# B&R Automation Studio project PO3
Automation Studio 4.5.2.102

## Configuration Real

### Hardware
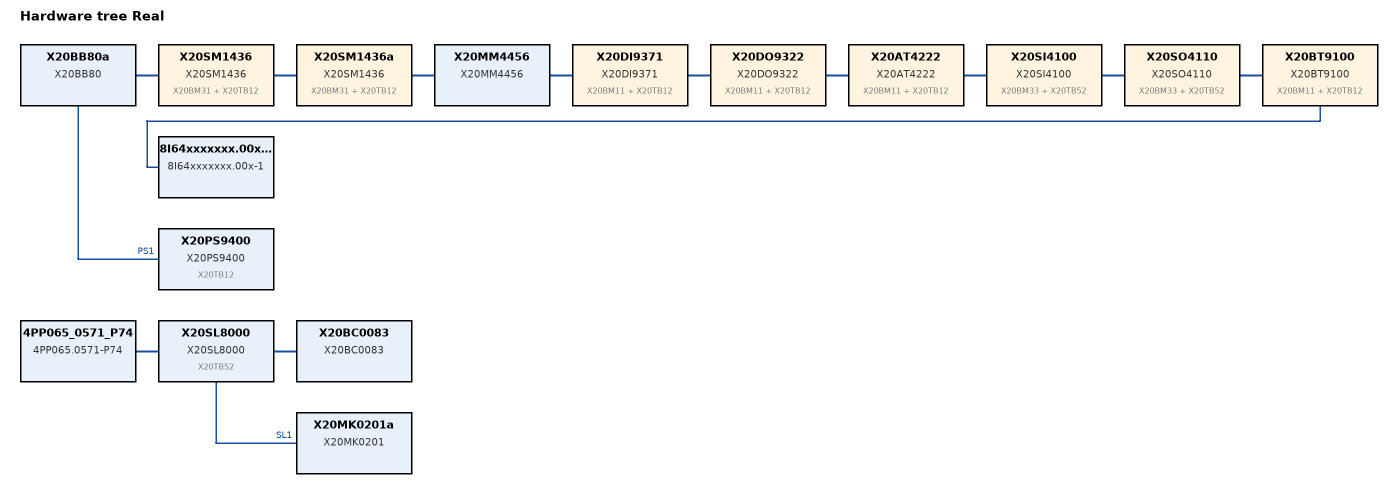
```
4PP065_0571_P74 : 4PP065.0571-P74 v1.1.2.0
  Connector IF4:
    EplInterfaceRedundant = 0
    EplEthInterfaceRedundant = 0
  Connector IF5:
    ActivateDevice = 1
    Mode = Manual
    InternetAddress = 10.0.1.10
    SubnetMask = 255.255.255.0
  ConfigurationID = LabBR
  TimerDeviceType = EPLX2X
  TimerDevice = 4PP065_0571_P74.IF4
  TaskClassIdleTime = 2000
  Cyclic1Duration = 2000
  Cyclic1Tolerance = 0
  Cyclic1Output = 1
  Cyclic3Tolerance = 0
  VcObjectName = Visu
8I64xxxxxxx.00x-1 : 8I64xxxxxxx.00x-1 v1.3.9.1  [X2X1 -> X20BT9100.X2X1 [Cable Type=X2XCable, Length=10, Version=1.0.0.2]]
  BothEndSwitchesAreNormallyOpen_r1 = on
  QuickStopIsNormallyOpen_r1 = on
X20AT4222 : X20AT4222 v1.2.3.0  [SS1 -> X20TB12f.SS; SL -> X20BM11c.SL1]
X20BB80a : X20BB80 v1.0.2.0
X20BC0083 : X20BC0083 v2.7.0.0  [PLK1 -> X20SL8000.PLK2 (NodeNumber=2) [Cable Type=PowerlinkCable, Length=10, Version=1.0.0.2]; SL -> X20BB80a.SL1]
X20BM11a : X20BM11 v1.0.0.1  [X2X1 -> X20MM4456.X2X2]
X20BM11b : X20BM11 v1.0.0.1  [X2X1 -> X20BM11a.X2X2]
X20BM11c : X20BM11 v1.0.0.1  [X2X1 -> X20BM11b.X2X2]
X20BM11d : X20BM11 v1.0.0.1  [X2X1 -> X20BM33b.X2X2]
X20BM31a : X20BM31 v1.0.0.1  [X2X1 -> X20BB80a.IF1]
X20BM31b : X20BM31 v1.0.0.1  [X2X1 -> X20BM31a.X2X2]
X20BM33a : X20BM33 v1.0.0.4  [X2X1 -> X20BM11c.X2X2]
X20BM33b : X20BM33 v1.0.0.4  [X2X1 -> X20BM33a.X2X2]
X20BT9100 : X20BT9100 v1.0.3.0  [SS1 -> X20TB12g.SS; SL -> X20BM11d.SL1]
X20DI9371 : X20DI9371 v1.0.2.0  [SS1 -> X20TB12d.SS; SL -> X20BM11a.SL1]
X20DO9322 : X20DO9322 v1.0.3.0  [SS1 -> X20TB12e.SS; SL -> X20BM11b.SL1]
X20MK0201a : X20MK0201 v1.0.0.0  [SL -> X20SL8000.SL1]
X20MM4456 : X20MM4456 v1.1.5.0  [X2X1 -> X20BM31b.X2X2]
X20PS9400 : X20PS9400 v1.0.2.4  [SS1 -> X20TB12b.SS; PS -> X20BB80a.PS1]
X20SI4100 : X20SI4100 v1.10.1.1  [SS1 -> X20TB52b.SS; SL -> X20BM33a.SL1]
X20SL8000 : X20SL8000 v1.6.5.1  [PLK1 -> 4PP065_0571_P74.IF4 (NodeNumber=1) [Cable Type=PowerlinkCable, Length=10, Version=1.0.0.2]; PLK2 -> X20BC0083.PLK1 (NodeNumber=1) [Cable Type=PowerlinkCable, Length=10, Version=1.0.0.2]; SS1 -> X20TB52a.SS]
  SafeProject = SafeLOGIC-1
X20SM1436 : X20SM1436 v1.4.2.1  [SS1 -> X20TB12a.SS; SL -> X20BM31a.SL1]
X20SM1436a : X20SM1436 v1.4.2.1  [SS1 -> X20TB12c.SS; SL -> X20BM31b.SL1]
X20SO4110 : X20SO4110 v1.10.1.1  [SS1 -> X20TB52c.SS; SL -> X20BM33b.SL1]
  SafeLogicID = 2
  SafeModuleID = 3
X20TB12a : X20TB12 v1.0.0.0
X20TB12b : X20TB12 v1.0.0.0
X20TB12c : X20TB12 v1.0.0.0
X20TB12d : X20TB12 v1.0.0.0
X20TB12e : X20TB12 v1.0.0.0
X20TB12f : X20TB12 v1.0.0.0
X20TB12g : X20TB12 v1.0.0.0
X20TB52a : X20TB52 v1.0.0.1
X20TB52b : X20TB52 v1.0.0.1
X20TB52c : X20TB52 v1.0.0.1
```

### IoMap.iom - 4PP065_0571_P74/IoMap.iom
```iecst
VAR_CONFIG
	Cyclic#1.gAxis03_DrvIf.iLifeCnt AT %IB."8I64xxxxxxx.00x-1".SDC_LifeCnt;
	Cyclic#1.gAxis03_DrvIf.iDrvOK AT %IX."8I64xxxxxxx.00x-1".ETAD_Input_Bool_02;
	Cyclic#1.gAxis03_DrvIf.oSetTime AT %QW."8I64xxxxxxx.00x-1".SDC_SetTime;
	Cyclic#1.gAxis03_DrvIf.oSetPos AT %QW."8I64xxxxxxx.00x-1".LFRD_Output;
	Cyclic#1.gAxis03_DiDoIf.iLifeCntDriveReady AT %IB."8I64xxxxxxx.00x-1".SDC_LifeCnt;
	Cyclic#1.gAxis03_DiDoIf.iLifeCntDriveEnable AT %IB."8I64xxxxxxx.00x-1".SDC_LifeCnt;
	Cyclic#1.gAxis03_DiDoIf.oDriveEnable AT %QX."8I64xxxxxxx.00x-1".CMDD_Output_Bool_00;
	Cyclic#1.gAxis03_ModuleOk AT %QX."8I64xxxxxxx.00x-1".CMDD_Output_Bool_01;
	Cyclic#1.gAxis03_ModuleOk AT %QX."8I64xxxxxxx.00x-1".CMDD_Output_Bool_02;
	Cyclic#1.gAxis03_ModuleOk AT %IX."8I64xxxxxxx.00x-1".ModuleOk;
	Cyclic#1.gAxis03_DiDoIf.oDriveEnable AT %QX."8I64xxxxxxx.00x-1".CMDD_Output_Bool_03;
	Cyclic#1.gAxis03_DiDoIf.iDriveReady AT %IX."8I64xxxxxxx.00x-1".ETAD_Input_Bool_02;
	::SDCAxisCtr:pwm_period AT %QW."X20MM4456".PeriodDurationPWM;
	::SDCAxisCtr:coil_pwm_value AT %QW."X20MM4456".PulseWidthCurrentPWM04;
	::SDCAxisCtr:axis_X.pwm_value AT %QW."X20MM4456".PulseWidthCurrentPWM01;
	::SDCAxisCtr:axis_X.reset_error AT %QX."X20MM4456".ClearError01;
	::SDCAxisCtr:axis_X.reset_counter AT %QX."X20MM4456".ResetCounter01;
	::SDCAxisCtr:axis_X.counter AT %IW."X20MM4456".Counter01;
	::SDCAxisCtr:coil_powered AT %IX."X20DI9371".DigitalInput01;
	::SDCAxisCtr:axis_X.endswitch_a_reached AT %IX."X20MM4456".StatusInput03;
	::SDCAxisCtr:axis_X.endswitch_b_reached AT %IX."X20MM4456".StatusInput04;
	::SDCAxisCtr:posEnable.enable AT %IX."X20DI9371".DigitalInput02; (*Insert your comment here...*)
	::SDCAxisCtr:posEnableRight.enable AT %IX."X20DI9371".DigitalInput03; (*Insert your comment here...*)
END_VAR
```

## Logical view

### Program Logical/Libraries/Library

#### FB_Axis.c
```c
#include <bur/plctypes.h>
#ifdef __cplusplus
	extern "C"
	{
#endif
	#include "Library.h"
#ifdef __cplusplus
	};
#endif
/* TODO: Add your comment here */
void FB_Axis(struct FB_Axis* inst)
{
	if (inst->endswitch_a_reached == 1 )
	{
		inst->dir = 1;
	}
	if (inst->endswitch_b_reached == 1 )
	{
		inst->dir = 0;
	}

	if(inst->dir == 1)
	{
		//inst->reset_counter = 0;
		inst->u = -inst->u;
		inst->pwm_value = (inst->u/24.0) * 32767;
	}
	if(inst->dir == 0)
	{
		//inst->reset_counter = 0;
		inst->pwm_value = (inst->u/24.0) * 32767;
	}
	if (inst->i == 1000)
	{
		inst->speed = (inst->counter - inst->last_counter)/2;
		inst->last_counter = inst->counter;
		inst->i = 0;
	}
	inst->spid = inst->speed;
	inst->i++;
}
```

### Program Logical/SDCAxisCtrl_X

#### Variables.var
```iecst
VAR
	min_task : INT := 7000;
	desired_speed : INT := 0;
	axis_X : FB_Axis;
	coil_powered : BOOL := FALSE;
	coil_pwm_value : {REDUND_UNREPLICABLE} INT := 200;
	fb_controller : FB_Controller;
	pwm_period : {REDUND_UNREPLICABLE} UINT := 200;
	Already_Homed : BOOL := FALSE;
	k : INT := 0;
	reset : BOOL := FALSE;
	posEnable : Pos := (0);
	posEnableRight : Pos := (0);
END_VAR
```

#### Main.c
```c
#include <bur/plctypes.h>

#ifdef _DEFAULT_INCLUDES
#include <AsDefault.h>
#endif

/* void increase_counters(void);
void Homing(void);
*/

void _INIT ProgramInit(void)
{

	//Устанваливаем типы SDC модулей
	AxisX_HW.EncIf1_Typ = ncSDC_ENC16;
	AxisX_HW.DiDoIf_Typ = ncSDC_DIDO;
	AxisX_HW.DrvIf_Typ = ncSDC_DRVSERVO16;

	//Устанавливаем имена переменных
	strcpy(AxisX_HW.EncIf1_Name, "AxisX_EncIf");
	strcpy(AxisX_HW.DrvIf_Name, "AxisX_DrvIf");
	strcpy(AxisX_HW.DiDoIf_Name, "AxisX_DiDoIf");

	//Устанавливаем входы готовности и нормальной работы
	AxisX_EncIf.iEncOK = 1;
	AxisX_DrvIf.iDrvOK = 1;
	AxisX_DrvIf.iStatusEnable = 1;
	AxisX_DiDoIf.iDriveReady = 1;

	fb_regulator.dt = 0.002;
	fb_regulator.k_i = 0.16;
	fb_regulator.k_p = 0.0064;
	fb_regulator.max_abc_value = 24.0;

	pwm_period = 200;
}

void _CYCLIC ProgramCyclic(void)
{
	if (posEnable.enable) {
	//	axis_X.endswitch_a_reached = 1;
		AxisX_DrvIf.oSetPos = -10000;
	} else if (posEnableRight.enable) {
		AxisX_DrvIf.oSetPos = 10000;
	}
	increase_counters();
	AxisX_EncIf.iActTime = (INT)AsIOTimeCyclicStart();
	iPosHwEnd = axis_X.endswitch_a_reached;
	iNegHwEnd = axis_X.endswitch_b_reached;

	if(coil_powered == 1)
	{
		if(!Already_Homed)
		{
			Homing();
		}
		else
		{
			increase_counters();
			axis_X.reset_counter = 0;
			FB_Axis(&axis_X);
			coil_pwm_value = 32767;
			iPosHwEnd = axis_X.endswitch_a_reached;
			iNegHwEnd = axis_X.endswitch_b_reached;
			FB_Axis(&axis_X);

			fb_regulator.e = (AxisX_DrvIf.oSetPos*10)  - axis_X.speed;//oSetPos;
			FB_Regulator(&fb_regulator);

			axis_X.u = fb_regulator.u ;
			FB_Axis(&axis_X);}
	}
	else
	{
		coil_pwm_value = 0;
		fb_regulator.e = 0 ;
		FB_Regulator(&fb_regulator);
		axis_X.u = 0;
		FB_Axis(&axis_X);

	}
	// COUNTER1 = axis_X.counter

	//COUNTER2 += axis_X.counter - COUNTER1;

}

void increase_counters(void)
{

	AxisX_EncIf.iLifeCnt++;
	AxisX_DiDoIf.iLifeCntDriveEnable++;
	AxisX_DiDoIf.iLifeCntDriveReady++;
	AxisX_DiDoIf.iLifeCntNegHwEnd++;
	AxisX_DiDoIf.iLifeCntPosHwEnd++;
	AxisX_DiDoIf.iLifeCntReference++;
	AxisX_DrvIf.iLifeCnt++;

}

void Homing(void)
{
	increase_counters();
	coil_pwm_value = 32767;
	iPosHwEnd = axis_X.endswitch_a_reached;
	iNegHwEnd = axis_X.endswitch_b_reached;
	FB_Axis(&axis_X);

	fb_regulator.e = (AxisX_DrvIf.oSetPos * 10) - axis_X.speed;//oSetPos;
	FB_Regulator(&fb_regulator);

	axis_X.u = fb_regulator.u ;
	FB_Axis(&axis_X);
	if (iPosHwEnd)
	{
		coil_pwm_value = 0;
		fb_regulator.e = 0;
		FB_Regulator(&fb_regulator);
		axis_X.u = 0;
		FB_Axis(&axis_X);
		axis_X.reset_counter = 1;
		FB_Axis(&axis_X);
		if(k == 200)
		{
			Already_Homed = 1;
			FB_Axis(&axis_X);
		}
		k++;

	}
}

void _EXIT ProgramExit(void)
{
	// Insert code here

}
```
